FUNCTION_BLOCK TM_DI16 (* Extracted Composite Function Block Type *)
  (* Standard: 61499-2 *)
  (* Version 25/02/2026 *)
  PACKAGE Hidryco.HidrycoLib;
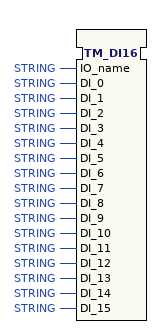
  VAR_INPUT
    IO_name : STRING;
    DI_0 : STRING;
    DI_1 : STRING;
    DI_2 : STRING;
    DI_3 : STRING;
    DI_4 : STRING;
    DI_5 : STRING;
    DI_6 : STRING;
    DI_7 : STRING;
    DI_8 : STRING;
    DI_9 : STRING;
    DI_10 : STRING;
    DI_11 : STRING;
    DI_12 : STRING;
    DI_13 : STRING;
    DI_14 : STRING;
    DI_15 : STRING;
  END_VAR
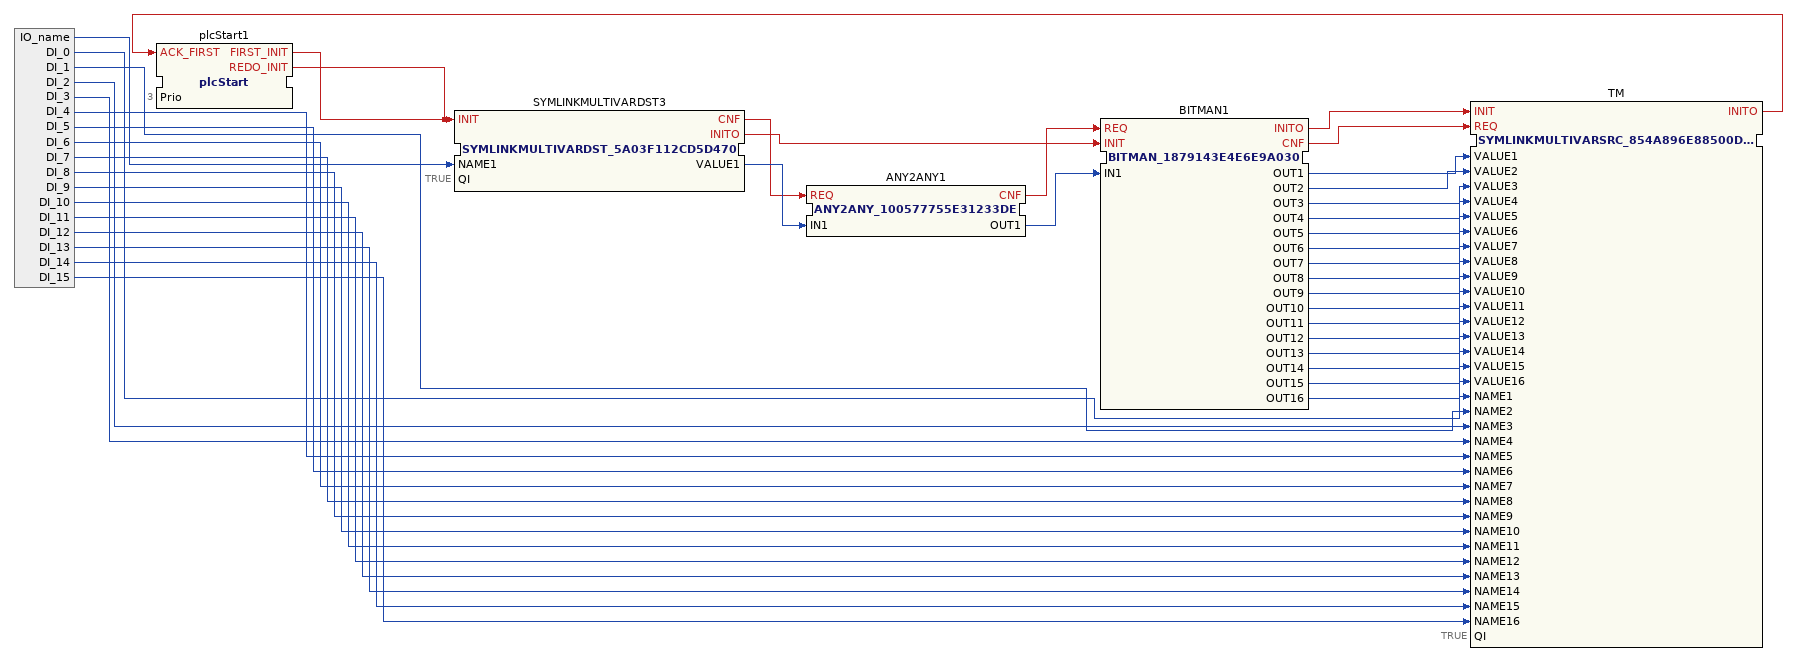
  FBS
    BITMAN1 : BITMAN_1879143E4E6E9A030; {SET_ATTRIBUTE(Configuration.GenericFBType.InterfaceParams, Runtime.Standard#CNTIN:=1;CNTOUT:=16;IN${CNTIN$}:WORD;OUT${CNTOUT$}:BOOL,BOOL,BOOL,BOOL,BOOL,BOOL,BOOL,BOOL,BOOL,BOOL,BOOL,BOOL,BOOL,BOOL,BOOL,BOOL)}
    SYMLINKMULTIVARDST3 : SYMLINKMULTIVARDST_5A03F112CD5D470(QI := TRUE); {SET_ATTRIBUTE(Configuration.GenericFBType.InterfaceParams, Runtime.System#I:=1;VALUE${I$}:INT)}
    ANY2ANY1 : ANY2ANY_100577755E31233DE; {SET_ATTRIBUTE(Configuration.GenericFBType.InterfaceParams, Runtime.Standard#CNT:=1;IN${CNT$}:INT;OUT${CNT$}:WORD)}
    TM : SYMLINKMULTIVARSRC_854A896E88500D19(QI := TRUE); {SET_ATTRIBUTE(Configuration.GenericFBType.InterfaceParams, Runtime.System#I:=16;VALUE${I$}:BOOL,BOOL,BOOL,BOOL,BOOL,BOOL,BOOL,BOOL,BOOL,BOOL,BOOL,BOOL,BOOL,BOOL,BOOL,BOOL)}
    plcStart1 : plcStart(Prio := 3);
  END_FBS
  EVENT_CONNECTIONS
    SYMLINKMULTIVARDST3.CNF TO ANY2ANY1.REQ;
    ANY2ANY1.CNF TO BITMAN1.REQ;
    SYMLINKMULTIVARDST3.INITO TO BITMAN1.INIT;
    BITMAN1.INITO TO TM.INIT;
    BITMAN1.CNF TO TM.REQ;
    plcStart1.FIRST_INIT TO SYMLINKMULTIVARDST3.INIT;
    plcStart1.REDO_INIT TO SYMLINKMULTIVARDST3.INIT;
    TM.INITO TO plcStart1.ACK_FIRST;
  END_CONNECTIONS
  DATA_CONNECTIONS
    SYMLINKMULTIVARDST3.VALUE1 TO ANY2ANY1.IN1;
    ANY2ANY1.OUT1 TO BITMAN1.IN1;
    BITMAN1.OUT1 TO TM.VALUE1;
    BITMAN1.OUT2 TO TM.VALUE2;
    BITMAN1.OUT3 TO TM.VALUE3;
    BITMAN1.OUT4 TO TM.VALUE4;
    BITMAN1.OUT5 TO TM.VALUE5;
    BITMAN1.OUT6 TO TM.VALUE6;
    BITMAN1.OUT7 TO TM.VALUE7;
    BITMAN1.OUT8 TO TM.VALUE8;
    BITMAN1.OUT9 TO TM.VALUE9;
    BITMAN1.OUT10 TO TM.VALUE10;
    BITMAN1.OUT11 TO TM.VALUE11;
    BITMAN1.OUT12 TO TM.VALUE12;
    BITMAN1.OUT13 TO TM.VALUE13;
    BITMAN1.OUT14 TO TM.VALUE14;
    BITMAN1.OUT15 TO TM.VALUE15;
    BITMAN1.OUT16 TO TM.VALUE16;
    IO_name TO SYMLINKMULTIVARDST3.NAME1;
    DI_0 TO TM.NAME1;
    DI_1 TO TM.NAME2;
    DI_2 TO TM.NAME3;
    DI_3 TO TM.NAME4;
    DI_4 TO TM.NAME5;
    DI_5 TO TM.NAME6;
    DI_6 TO TM.NAME7;
    DI_7 TO TM.NAME8;
    DI_8 TO TM.NAME9;
    DI_9 TO TM.NAME10;
    DI_10 TO TM.NAME11;
    DI_11 TO TM.NAME12;
    DI_12 TO TM.NAME13;
    DI_13 TO TM.NAME14;
    DI_14 TO TM.NAME15;
    DI_15 TO TM.NAME16;
  END_CONNECTIONS
END_FUNCTION_BLOCK
